{attribute addProperty BoxType "EJ2521-0224-0016"}
{attribute addProperty Id "Sel_Ack_End_counterBIT10.1251Ramp_activeBIT10.1252ErrorBIT10.1257Sync_errorBIT10.12514TxPDO_ToggleBIT10.12516"}
{attribute addProperty CRC "813189523"}
{attribute addProperty SizeInBites "16"}
{attribute addProperty SizeInBytes "2"}
TYPE Status_30784993 :
STRUCT
	{attribute addProperty Name "Sel_Ack_End_counter"}
	Sel_Ack_End_counter : BOOL;
	{attribute addProperty Name "Ramp_active"}
	Ramp_active : BOOL;
	{attribute 'hide'}
	reserve_1_BIT_0 : BOOL;
	{attribute 'hide'}
	reserve_1_BIT_1 : BOOL;
	{attribute 'hide'}
	reserve_1_BIT_2 : BOOL;
	{attribute 'hide'}
	reserve_1_BIT_3 : BOOL;
	{attribute addProperty Name "Error"}
	Error : BOOL;
	{attribute 'hide'}
	reserve_2_BIT_0 : BOOL;
	{attribute 'hide'}
	reserve_2_BIT_1 : BOOL;
	{attribute 'hide'}
	reserve_2_BIT_2 : BOOL;
	{attribute 'hide'}
	reserve_2_BIT_3 : BOOL;
	{attribute 'hide'}
	reserve_2_BIT_4 : BOOL;
	{attribute 'hide'}
	reserve_2_BIT_5 : BOOL;
	{attribute addProperty Name "Sync_error"}
	Sync_error : BOOL;
	{attribute 'hide'}
	reserve_3 : BOOL;
	{attribute addProperty Name "TxPDO_Toggle"}
	TxPDO_Toggle : BOOL;
END_STRUCT
END_TYPE

(* stored: Version 1.2.0.0, ProductVersion 3.1.4024.9
   DUT Status_30784993: Id {d7090b00-c3f7-422a-8fd6-4413e7c2feb7} *)
